(* CoDeSys 2.3.9.59 project: ads.pro *)
(* Libraries: TcBase.lib 14.5.09 11:14:08, TcSystem.lib*7.6.16 10:01:22, TwinCAT\Plc\Lib\TcUtilities.lib 3.2.16 15:08:58, STANDARD.LIB 5.6.98 11:03:02 *)

(* Task configuration *)
TASK Standard (PRIORITY := 0, INTERVAL := T#4ms);
	MAIN
END_TASK

(* Global variable list: Global_Variables *)
VAR_GLOBAL
	(* variable test  *)
	junit_bit					:BOOL;
	junit_int8					:SINT;
	junit_int16				:INT;
	junit_int32				:DINT;
	junit_uint8				:BYTE;
	junit_uint16				:WORD;
	junit_uint32				:DWORD;
	junit_real32				:REAL;
	junit_real64				:LREAL;
	junit_string				:STRING(100);

	(* loader test  *)
	junit_array_small			:ARRAY[0..2] OF INT;
	junit_array_simple			:ARRAY[0..2, 2..4, 4..6] OF INT;
	junit_array_complex		:ARRAY[0..2, 4..8] OF fb_junit;
	junit_function_block		:fb_junit;
	juint_struct				:junit_st;

	(* problem *)
	junit_time					:TIME;
	juinit_p_simple			:POINTER TO LREAL;
	juinit_p_complex			:POINTER TO junit_st;
	juinit_p_complex_array 	:POINTER TO ARRAY [0..2] OF junit_st;
END_VAR

VAR_GLOBAL CONSTANT
	junit_c			:INT := 10;
END_VAR

(* Data type *)
TYPE junit_st :
STRUCT
	b_value		:BOOL;
	st_value		:TON;
END_STRUCT
END_TYPE

(* POU main, ST *)
PROGRAM main
VAR
	l_fb_unit	:fb_junit;

	l_ams_port		:UDINT:=AMSPORT_R3_SYSSERV;
	l_index_group	:UDINT:=SYSTEMSERVICE_ENUMREMOTE;
	l_index_offset		:UDINT;
	l_read_type		: ST_AmsRouteSystemEntry;
	l_read_size		:UDINT;
END_VAR
l_read_size	:= SIZEOF( l_read_type );
END_PROGRAM

(* POU fb_junit, ST *)
FUNCTION_BLOCK fb_junit
VAR_INPUT
	input	:BOOL;
END_VAR

VAR_OUTPUT
	output	:LREAL;
END_VAR

VAR
	internal_structure			:junit_st;
	internal_primitive			:INT;
	internal_primitive_array		:ARRAY [0..2] OF BOOL;
	internal_structure_array		:ARRAY [1..3] OF junit_st;
END_VAR
;
END_FUNCTION_BLOCK

(* POU p_enum_route_entries, ST *)
PROGRAM p_enum_route_entries
VAR
   fbEnum : FB_EnumRouteEntry := ( sNetID := '', tTimeout := T#5s );
    bEnum  : BOOL := TRUE;
    nState : BYTE := 0;
    sInfo  : T_MaxString;
END_VAR
CASE nState OF
    0:
    IF bEnum THEN (* flag set ? *)
        bEnum := FALSE; (* reset flag *)
        fbEnum.eCmd := eEnumCmd_First; (* enum first entry *)
        nState := 1;
    END_IF

    1: (* enum one entry *)
    fbEnum( bExecute := FALSE );
    fbEnum( bExecute := TRUE );
    nState := 2;

    2: (* wait until function block not busy *)
    fbEnum( bExecute := FALSE );
    IF NOT fbEnum.bBusy THEN
        IF NOT fbEnum.bError THEN
            IF NOT fbEnum.bEOE THEN
                sInfo := CONCAT( 'Name: ', fbEnum.stRoute.sName );
                sInfo := CONCAT( sInfo, ' Address: ' );
                sInfo := CONCAT( sInfo, fbEnum.stRoute.sAddress );
                sInfo := CONCAT( sInfo, ' Transport: ' );
                sInfo := CONCAT( sInfo, ROUTETRANSPORT_TO_STRING( fbEnum.stRoute.eTransport ) );
                ADSLOGSTR( ADSLOG_MSGTYPE_HINT OR ADSLOG_MSGTYPE_LOG, 'ROUTE INFO: %s', sInfo );
                    fbEnum.eCmd := eEnumCmd_Next; (* enum next entry *)
                nState := 1;
            ELSE (* no more route entries *)
                nState := 0;
            END_IF
        ELSE (* log error *)
            ADSLOGSTR( ADSLOG_MSGTYPE_ERROR OR ADSLOG_MSGTYPE_LOG, 'FB_EnumRouteEntry error:%s', DWORD_TO_HEXSTR( fbEnum.nErrID, 0, FALSE ) );
            nState := 0;
        END_IF
    END_IF
END_CASE
END_PROGRAM

(* POU p_juinit, ST *)
PROGRAM p_juinit
VAR
	l_ams_port 			:INT;
	l_idxGrp				:UDINT;
	l_size				:INT;
	l_size_entry			:ST_AmsRouteSystemEntry;

	l_FB_EnumRouteEntry 	:FB_EnumRouteEntry;
	l_sNetID				:STRING := '127.0.0.1.1.1';
	l_eCmd      			:E_EnumCmdType;
	l_b_busy				:BOOL;
	l_b_error				:BOOL;
	l_ud_nErrID			:UDINT;
	l_bEOE				:BOOL;
	l_route_data			:ST_AmsRouteEntry;
END_VAR
	l_ams_port 	:= AMSPORT_R3_SYSSERV;
	l_idxGrp		:= SYSTEMSERVICE_ENUMREMOTE;
	l_size		:= SIZEOF(l_size_entry);

	p_enum_route_entries;
END_PROGRAM
